// TIA Portal V20 export
// export: Created 2026-04-11T06:02:30.1157232Z, ExportSetting WithDefaults, DisplayName Totally Integrated Automation Portal, DisplayVersion V20, DisplayName TIA Portal Openness, DisplayVersion V20, DisplayName TIA Portal Version Control Interface, DisplayVersion V20, DisplayName STEP 7 Professional, DisplayVersion V20, DisplayName STEP 7 Safety, DisplayVersion V20, DisplayName WinCC Basic/Comfort/Advanced, DisplayVersion V20, DisplayName WinCC Unified, DisplayVersion V20
TYPE "udtError_MotorStarterET200"
// stored: IsFailsafeCompliant false
   STRUCT
      NoSignalForward { ExternalWritable := 'False'} : Bool;   // No signal from forward command
      NoSignalReverse { ExternalWritable := 'False'} : Bool;   // No signal from reverse command
      MotorNotStopped { ExternalWritable := 'False'} : Bool;   // Motor doesn't stop
      GroupWarning { ExternalWritable := 'False'} : Bool;   // Group Warning
      GroupFault { ExternalWritable := 'False'} : Bool;   // Group Fault
      CurrentLimitTripping { ExternalWritable := 'False'} : Bool;   // Current Limit Tripping
      ResidualCurrentDetected { ExternalWritable := 'False'} : Bool;   // Residual Current Detected
      AsymmetryDetected { ExternalWritable := 'False'} : Bool;   // Asymmetry Detected
      OverTemperature { ExternalWritable := 'False'} : Bool;   // Over Temperature
      ThermalMotorModelOverload { ExternalWritable := 'False'} : Bool;   // Thermal Motor Model Overload
   END_STRUCT;
END_TYPE
